// TIA Portal project "S7-1500 için JMP-JMPN-LABEL Komutu" (V18)

(* hardware
DEVICE "S7-1500/ET200MP station_1"  S7-1500 station
   slot 0: "Rail_0"  Rack  6ES7 590-1***0-0AA0
   slot 1: "PLC_1"  CPU 1512C-1 PN  6ES7 512-1CK00-0AB0  V2.8
      slot 3: "CPU display_1"  6ES7591-1AA00-0AA0
      slot 32768: "PROFINET interface_1"  X1
         slot 32769: "Port_1"  X1 P1
         slot 32770: "Port_2"  X1 P2
      slot 34817: "Virtual CP interface port_1"  Virtual CP interface port  Virtual CP interface port
*)

// ===== PLC "PLC_1"  CPU 1512C-1 PN =====

VAR_GLOBAL   // PLC tag table "Default tag table"
   "Tag_1" AT %I0.0 : Bool;
   "Tag_2" AT %MW10 : Int;
   "Tag_3" AT %Q0.0 : Bool;
   "Tag_4" AT %I0.1 : Bool;
   "Tag_5" AT %Q0.1 : Bool;
   "Tag_6" AT %MW11 : Int;
   "Tag_7" AT %MW12 : Int;
   "Tag_8" AT %MW13 : Int;
   "Tag_9" AT %MW14 : Int;
   "Tag_10" AT %I0.2 : Bool;
   "Tag_11" AT %I0.3 : Bool;
   "Tag_12" AT %MW5 : Word;
   "Tag_13" AT %MW6 : Word;
   "Tag_14" AT %MW8 : Word;
   "Tag_15" AT %MW19 : Word;
   "Tag_16" AT %MW9 : Word;
END_VAR

// folder: System blocks/Program resources

DATA_BLOCK "IEC_Counter_0_DB"   // DB1
{ S7_Optimized_Access := 'TRUE' }
AUTHOR : Simatic
FAMILY : IEC
NAME : CNTR
VERSION : 1.0
// stored: InstanceOfName IEC_COUNTER
"IEC_COUNTER"
BEGIN
END_DATA_BLOCK

// folder: (top level)

ORGANIZATION_BLOCK "Main"   // OB1, LAD, ProgramCycle
TITLE = "Main Program Sweep (Cycle)"
{ S7_Optimized_Access := 'TRUE' }
VERSION : 0.1
   VAR_INPUT
      Initial_Call : Bool;   // Initial call of this OB
      Remanence : Bool;   // =True, if remanent data are available
   END_VAR
BEGIN

REGION Network 1: JMP önündeki kontak 1 olunca sıçrama yapar.
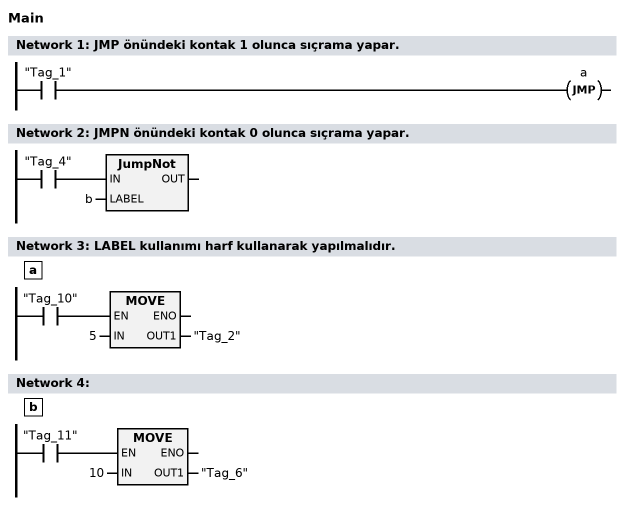
   RUNG wire#powerrail
      Contact( "Tag_1" )
      JumpCoil( a )
   END_RUNG
   // the same network as SCL:
   IF "Tag_1" THEN GOTO a; END_IF;
END_REGION

REGION Network 2: JMPN önündeki kontak 0 olunca sıçrama yapar.
   // no SCL statement known for JumpNot: written as a call
   JumpNot(in := "Tag_4", label := b);
END_REGION

REGION Network 3: LABEL kullanımı harf kullanarak yapılmalıdır.
   Label( a )
   RUNG wire#powerrail
      Contact( "Tag_10" )
      Move(in := 5, out1 => "Tag_2")
   END_RUNG
   // the same network as SCL:
   a:
   IF "Tag_10" THEN "Tag_2" := 5; END_IF;
END_REGION

REGION Network 4
   Label( b )
   RUNG wire#powerrail
      Contact( "Tag_11" )
      Move(in := 10, out1 => "Tag_6")
   END_RUNG
   // the same network as SCL:
   b:
   IF "Tag_11" THEN "Tag_6" := 10; END_IF;
END_REGION
END_ORGANIZATION_BLOCK